// LS Electric XG5000 project: 2022_03_02_지방3과제
// PLC NewPLC
// module base 0 slot 0: 입출력 모듈:XBC-DR32H (DC 24V 입력, 릴레이 출력 32점)
// module base 0 slot 1: 위치결정 모듈:XBF-PD02A (위치결정 펄스(LD)출력형, 2축)
// module base 0 slot 2: 출력 모듈:XBE-TN/TP16A (트랜지스터 출력, 16점 (싱크출력/소스출력))

PROGRAM 지방3과제레더 (task: 스캔 프로그램)

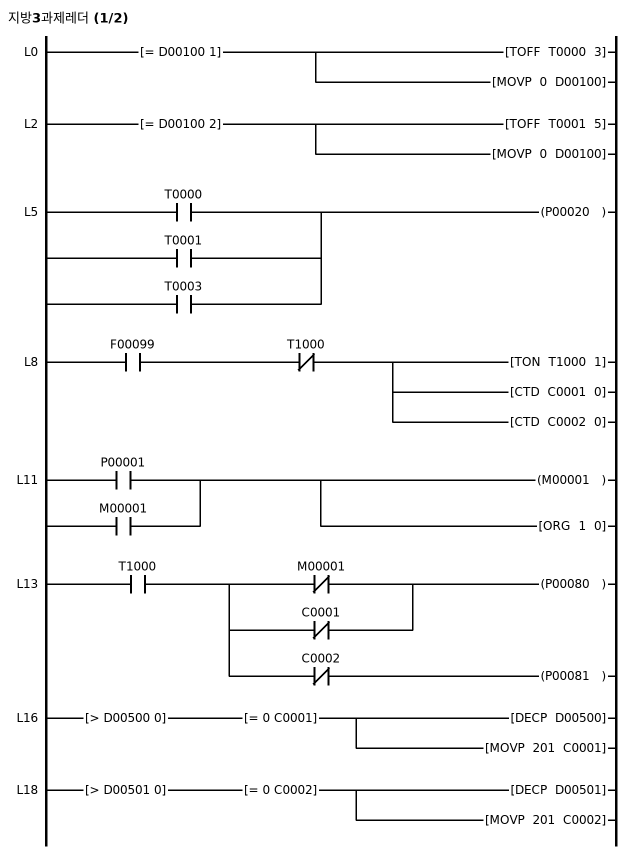
; L0
LOAD=     D00100 1
TOFF      T0000 3
MOVP      0 D00100
; L2
LOAD=     D00100 2
TOFF      T0001 5
MOVP      0 D00100
; L5
LOAD      T0000
OR        T0001
OR        T0003
OUT       P00020
; L8
LOAD      F00099
AND NOT   T1000
TON       T1000 1
CTD       C0001 0
CTD       C0002 0
; L11
LOAD      P00001
OR        M00001
OUT       M00001
ORG       1 0
; L13
LOAD      T1000
MPUSH
LOAD NOT  M00001
OR NOT    C0001
AND LOAD
OUT       P00080
MPOP
AND NOT   C0002
OUT       P00081
; L16
LOAD>     D00500 0
AND=      0 C0001
DECP      D00500
MOVP      201 C0001
; L18
LOAD>     D00501 0
AND=      0 C0002
DECP      D00501
MOVP      201 C0002

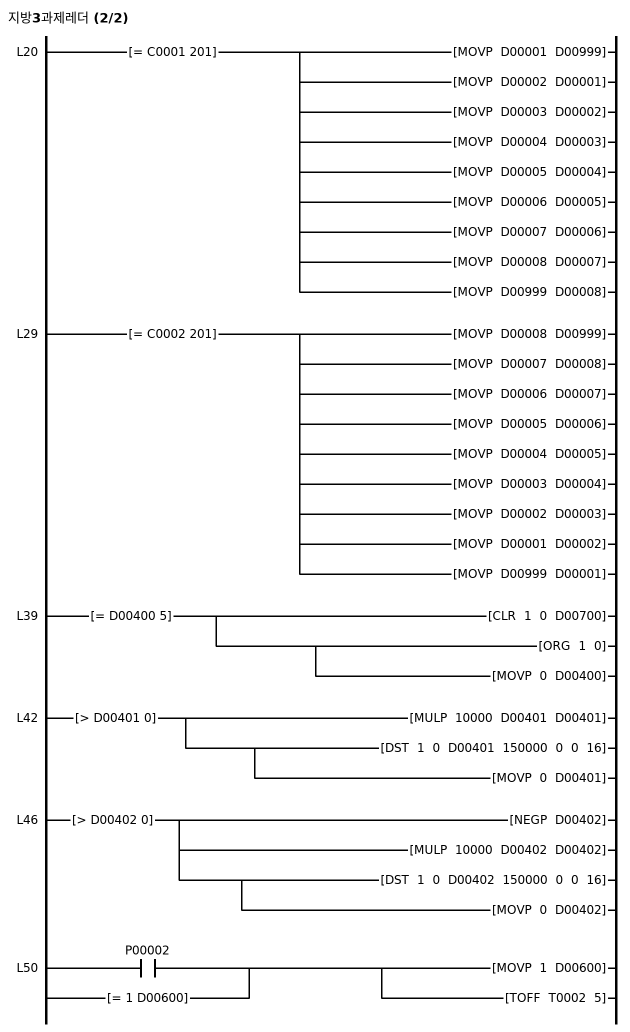
; L20
LOAD=     C0001 201
MOVP      D00001 D00999
MOVP      D00002 D00001
MOVP      D00003 D00002
MOVP      D00004 D00003
MOVP      D00005 D00004
MOVP      D00006 D00005
MOVP      D00007 D00006
MOVP      D00008 D00007
MOVP      D00999 D00008
; L29
LOAD=     C0002 201
MOVP      D00008 D00999
MOVP      D00007 D00008
MOVP      D00006 D00007
MOVP      D00005 D00006
MOVP      D00004 D00005
MOVP      D00003 D00004
MOVP      D00002 D00003
MOVP      D00001 D00002
MOVP      D00999 D00001
; L39
LOAD=     D00400 5
CLR       1 0 D00700
ORG       1 0
MOVP      0 D00400
; L42
LOAD>     D00401 0
MULP      10000 D00401 D00401
DST       1 0 D00401 150000 0 0 16
MOVP      0 D00401
; L46
LOAD>     D00402 0
NEGP      D00402
MULP      10000 D00402 D00402
DST       1 0 D00402 150000 0 0 16
MOVP      0 D00402
; L50
LOAD      P00002
OR=       1 D00600
MOVP      1 D00600
TOFF      T0002 5